PROGRAM RS232_Communication
VAR
	fbPcCom		: FB_SerialCom;
	
	(* exchange buffers with background communication with the PC COM port device *)
	RxBufferPcCom	: ComBuffer;	(* Receive data buffer; used with all receive function blocks *)
	TxBufferPcCom	: ComBuffer;	(* Transmit data buffer; used with all receive function blocks *)
END_VAR

(* background communication with the PC COM port device *)
BackgroundPcCOM(RxBufferPcCom:=RxBufferPcCom, TxBufferPcCom:=TxBufferPcCom);

(* Send and receive commands *)
fbPcCom(TxBuffer:=TxBufferPcCom, RxBuffer:=RxBufferPcCom);

END_PROGRAM

(* stored: Version 1.1.0.1, ProductVersion 3.1.4022.3
   POU RS232_Communication: Id {aef089b1-c7c5-479f-8336-a7bf9b8b2785}, SpecialFunc None *)
